Yaskawa INFORM job: OK_R2_O55B(90,0)KMOK.JBI

/JOB
//NAME OK_R2_O55B(90,0)KMOK
//POS
///NPOS 391,391,391,17,0,0
///TOOL 0
///POSTYPE PULSE
///PULSE
C00000=-9957,-80120,-66349,29251,62843,-41580
C00001=-130831,-56999,-52491,28072,65386,-40358
C00002=-127931,-24435,-32256,25248,67356,-37514
C00003=-126700,-19683,-26605,24973,66044,-37324
C00004=-125164,-19903,-26767,24398,65578,-36815
C00005=-126700,-19683,-26605,24973,66044,-37324
C00006=-126700,-19454,-24775,25160,65129,-37533
C00007=-126700,-19683,-26605,24973,66044,-37324
C00008=-126519,-14725,-22916,24857,66242,-37208
C00009=-126700,-19683,-26605,24973,66044,-37324
C00010=-127431,-22768,-30880,25062,67214,-37348
C00011=-129904,-26243,-35656,25771,69013,-37912
C00012=-103883,-33865,-42899,-26333,63628,-24210
C00013=-104076,-28068,-33208,-26929,60884,-23597
C00014=-104308,-24022,-28158,-27086,59888,-23435
C00015=-104293,-23807,-26929,-27261,59318,-23277
C00016=-104308,-24022,-28158,-27086,59888,-23435
C00017=-104568,-21372,-26276,-26919,59985,-23573
C00018=-104308,-24022,-28158,-27086,59888,-23435
C00019=-104359,-30091,-33838,-26967,60209,-23541
C00020=-104172,-35756,-40489,-26759,61329,-23752
C00021=-101371,-58624,-53351,-28997,58954,-21848
C00022=-130278,-21019,-10450,28766,57658,-40988
C00023=-127795,-16814,-4966,28257,55740,-40424
C00024=-124867,-3493,1682,21696,65206,-34879
C00025=-124867,-2956,3429,21830,64460,-35026
C00026=-124867,-3493,1682,21696,65206,-34879
C00027=-123403,-3637,1565,21295,64821,-34374
C00028=-124867,-3493,1682,21696,65206,-34879
C00029=-124781,112,4661,21670,65203,-34846
C00030=-126448,-16298,-3504,27965,54725,-40103
C00031=-127417,-18060,-5778,28164,55488,-40325
C00032=-129915,-24050,-16876,27962,59657,-40264
C00033=-103828,-30318,-23260,-29155,54504,-21694
C00034=-104023,-24208,-16094,-29514,53321,-21419
C00035=-104359,-18909,-9882,-29771,52240,-21236
C00036=-104359,-18502,-8615,-29989,51742,-21073
C00037=-104359,-18909,-9882,-29771,52240,-21236
C00038=-104548,-17165,-8596,-29647,52265,-21334
C00039=-104359,-18909,-9882,-29771,52240,-21236
C00040=-104284,-25793,-15917,-29738,52421,-21258
C00041=-104095,-31966,-23082,-29370,53571,-21532
C00042=-101389,-51580,-31391,-32519,50375,-19075
C00043=-130293,-20904,-10309,28779,57639,-41000
C00044=-127810,-16697,-4821,28272,55719,-40437
C00045=-124421,-5878,1074,22169,61673,-35261
C00046=-123293,-5978,993,21815,61369,-34862
C00047=-124421,-5878,1074,22169,61673,-35261
C00048=-124421,-5464,2370,22286,61130,-35375
C00049=-124421,-5878,1074,22169,61673,-35261
C00050=-124367,-3413,3070,22144,61694,-35234
C00051=-124421,-5878,1074,22169,61673,-35261
C00052=-127374,-17559,-5212,28177,55393,-40333
C00053=-129863,-23659,-16652,27928,59696,-40231
C00054=-104291,-30466,-23154,-28998,54219,-21823
C00055=-104471,-24344,-15984,-29365,53043,-21545
C00056=-104848,-18627,-9754,-29526,52126,-21437
C00057=-104848,-18034,-7918,-29844,51404,-21206
C00058=-104848,-18372,-8952,-29664,51809,-21336
C00059=-105025,-16673,-7696,-29545,51834,-21430
C00060=-104848,-18372,-8952,-29664,51809,-21336
C00061=-104541,-25679,-16044,-29572,52449,-21391
C00062=-104362,-31845,-23206,-29202,53599,-21667
C00063=-101422,-47913,-22789,-34118,47488,-17974
C00064=-130262,-20482,-9952,28769,57626,-40991
C00065=-127787,-16271,-4450,28267,55703,-40431
C00066=-125772,-1300,4566,24233,64800,-37238
C00067=-125099,-11874,382,27493,54175,-39643
C00068=-126165,-11734,491,27896,54532,-40029
C00069=-126165,-11290,1726,28071,54059,-40171
C00070=-126165,-11734,491,27896,54532,-40029
C00071=-126097,-9728,2048,27846,54574,-39985
C00072=-126165,-11734,491,27896,54532,-40029
C00073=-127493,-17714,-5356,28218,55441,-40373
C00074=-129987,-23980,-17397,27894,59998,-40203
C00075=-104210,-30109,-23029,-28998,54341,-21823
C00076=-104392,-23995,-15854,-29364,53158,-21544
C00077=-104664,-19137,-9875,-29681,52028,-21314
C00078=-104664,-18688,-8489,-29921,51485,-21138
C00079=-104664,-19137,-9875,-29681,52028,-21314
C00080=-104885,-17048,-8334,-29533,52061,-21432
C00081=-104664,-19137,-9875,-29681,52028,-21314
C00082=-104584,-25734,-15966,-29581,52368,-21386
C00083=-104406,-31905,-23130,-29210,53516,-21662
C00084=-101487,-56722,-46956,-29848,56320,-21116
C00085=-130260,-20245,-9571,28802,57525,-41018
C00086=-127787,-16027,-4057,28303,55600,-40460
C00087=-126397,-12024,-58,27921,54776,-40065
C00088=-126397,-11418,1630,28163,54132,-40255
C00089=-126397,-12024,-58,27921,54776,-40065
C00090=-125058,-12202,-195,27417,54327,-39580
C00091=-126397,-12024,-58,27921,54776,-40065
C00092=-126319,-9801,1666,27863,54821,-40014
C00093=-126397,-12024,-58,27921,54776,-40065
C00094=-127466,-17804,-5568,28181,55506,-40341
C00095=-129961,-24611,-19623,27616,60919,-39941
C00096=-104121,-29849,-22868,-29026,54402,-21800
C00097=-104306,-23738,-15686,-29392,53214,-21520
C00098=-104574,-18869,-9557,-29743,52009,-21266
C00099=-104574,-18451,-8267,-29970,51501,-21102
C00100=-104574,-18869,-9557,-29743,52009,-21266
C00101=-104772,-17011,-8185,-29613,52038,-21371
C00102=-104574,-18869,-9557,-29743,52009,-21266
C00103=-104605,-25690,-15920,-29574,52356,-21392
C00104=-101416,-53614,-36326,-31658,51963,-19708
C00105=-101416,-53614,-36326,-31658,51963,-19708
C00106=-113373,-19710,-23567,-5252,67661,-28636
C00107=-114752,-18608,-16975,3728,63450,-28918
C00108=-121641,-12158,-10795,16175,65821,-31343
C00109=-121641,-11553,-8404,16318,64706,-31501
C00110=-121642,-12221,-10110,16230,65385,-31404
C00111=-120492,-12233,-10119,15867,65157,-30993
C00112=-121644,-12965,-11195,16196,65660,-31365
C00113=-121703,-22742,-18426,16285,65120,-31465
C00114=-116423,-24349,-16589,8028,59581,-22849
C00115=-116462,-22943,-15594,8034,59695,-22855
C00116=-117089,-27968,-21523,8194,60813,-23017
C00117=-138257,-43921,-38980,29449,67834,19559
C00118=-154095,-44107,-36576,41026,64683,28586
C00119=-155372,-26710,-22710,49007,54658,45155
C00120=-156430,-13085,-10936,68207,72434,47480
C00121=-154097,-10834,-6257,68530,70189,47037
C00122=-153034,-8688,-2137,68930,68920,46537
C00123=-153034,-8230,-667,69164,68664,46234
C00124=-153034,-8688,-2137,68930,68920,46537
C00125=-152716,-7159,-923,68899,68723,46597
C00126=-153034,-8688,-2137,68930,68920,46537
C00127=-155527,-11962,-5672,68921,70786,46416
C00128=-157894,-14200,-10337,68577,73047,46860
C00129=-156589,-13315,-10824,68272,72466,47375
C00130=-154250,-11059,-6142,68601,70219,46932
C00131=-153110,-8549,-1740,68995,68901,46448
C00132=-153110,-8137,-433,69201,68672,46178
C00133=-153110,-8549,-1740,68995,68901,46448
C00134=-152772,-6933,-461,68963,68694,46512
C00135=-153110,-8549,-1740,68995,68901,46448
C00136=-155649,-11770,-5813,68871,70940,46483
C00137=-158013,-13984,-10461,68536,73200,46927
C00138=-156493,-13364,-11001,68241,72435,47426
C00139=-154155,-11109,-6321,68567,70188,46983
C00140=-153047,-8804,-2189,68941,68917,46522
C00141=-153047,-8341,-714,69171,68660,46216
C00142=-153047,-8804,-2189,68941,68917,46522
C00143=-152699,-7122,-856,68902,68699,46591
C00144=-153047,-8804,-2189,68941,68917,46522
C00145=-155528,-12235,-6032,68896,70818,46453
C00146=-157898,-14465,-10687,68556,73081,46895
C00147=-156404,-13719,-11255,68241,72365,47427
C00148=-154061,-11456,-6573,68567,70116,46985
C00149=-152978,-9293,-2613,68935,68873,46536
C00150=-152978,-8887,-1313,69141,68646,46265
C00151=-152978,-9293,-2613,68935,68873,46536
C00152=-152568,-7316,-1048,68891,68617,46616
C00153=-152978,-9293,-2613,68935,68873,46536
C00154=-155488,-12320,-6114,68891,70795,46461
C00155=-157860,-14552,-10769,68552,73058,46903
C00156=-156499,-13757,-11316,68244,72435,47421
C00157=-154155,-11502,-6641,68569,70186,46980
C00158=-152940,-8723,-2197,68919,68862,46557
C00159=-152940,-8321,-897,69127,68633,46287
C00160=-152940,-8723,-2197,68919,68862,46557
C00161=-152615,-7149,-950,68886,68660,46620
C00162=-152940,-8723,-2197,68919,68862,46557
C00163=-155527,-12441,-6175,68901,70811,46445
C00164=-157901,-14672,-10829,68562,73075,46886
C00165=-154973,1945,11064,69380,67800,43696
C00166=-153498,388,9750,69327,66810,43901
C00167=-151944,3598,13389,69509,65547,43839
C00168=-152901,-833,7436,68993,66712,44352
C00169=-153760,-1170,8451,69337,66987,43865
C00170=-150992,-308,10136,69473,64908,43968
C00171=-151435,4354,14125,69671,69854,43018
C00172=-151601,9028,18225,69679,74023,42144
C00173=-153599,495,9837,69084,71042,58093
C00174=-155601,2650,11659,69106,72383,57818
C00175=-155003,-799,3033,68136,69188,45300
C00176=-153529,-1129,5762,68693,67473,44668
C00177=-151691,2413,10794,69105,65750,44340
C00178=-152932,-1773,5149,68640,67090,44774
C00179=-153793,-2147,6130,68987,67361,44287
C00180=-151088,-288,8615,69107,65323,44406
C00181=-151404,3599,11904,69364,69896,43458
C00182=-151218,5876,13928,69450,72821,42839
C00183=-153630,-777,6611,68687,71576,58686
C00184=-155633,219,4703,68296,73580,59159
C00185=-154938,2214,11292,69379,67776,43700
C00186=-153465,658,9976,69326,66788,43906
C00187=-151970,3515,13352,69518,65553,43829
C00188=-152869,-564,7660,68991,66691,44357
C00189=-153727,-902,8674,69336,66964,43870
C00190=-151411,1015,11233,69490,65183,43915
C00191=-150298,-2919,8029,69467,64414,44045
C00192=-151641,9147,18309,69679,73942,42091
C00193=-153566,764,10064,69084,71020,58097
C00194=-155565,2919,11887,69107,72358,57821
C00195=-154990,1810,10950,69380,67812,43694
C00196=-153514,253,9637,69328,66822,43899
C00197=-151956,3103,12633,69423,65630,43940
C00198=-152917,-967,7324,68994,66723,44350
C00199=-153777,-1304,8340,69338,66998,43862
C00200=-151252,489,10575,69428,65130,44000
C00201=-151705,5965,15347,69658,70903,42778
C00202=-151762,10642,19506,69646,75062,41892
C00203=-153615,360,9724,69084,71054,58091
C00204=-155619,2515,11544,69106,72395,57816
C00205=-154955,2080,11178,69379,67788,43698
C00206=-153481,523,9864,69327,66799,43904
C00207=-152005,3278,13000,69479,65609,43868
C00208=-152885,-698,7548,68992,66701,44355
C00209=-153744,-1035,8563,69337,66975,43867
C00210=-151366,800,11018,69477,65161,43933
C00211=-151607,5013,14724,69679,69923,42916
C00212=-151807,11049,20057,69670,75075,41824
C00213=-153582,630,9951,69084,71031,58095
C00214=-155583,2785,11773,69106,72370,57820
C00215=-147758,2086,2374,31053,60988,58888
C00216=-133325,-38773,-33930,6315,58066,25890
C00217=-110400,-54315,-51528,-18458,56734,4707
C00218=-102274,-32558,-14872,-44027,37469,-32506
C00219=-105929,-26421,-10740,-41149,36164,-34321
C00220=-116067,-24319,-8645,-13286,26575,-50151
C00221=-116038,-24316,-8643,-13324,26580,-50130
C00222=-111352,-27223,-10659,-19551,27279,-46780
C00223=-103129,-25181,-9190,-38570,34106,-35952
C00224=-100769,-25035,-8960,-40367,35121,-34847
C00225=-99695,-24670,-8429,-41242,35512,-34306
C00226=-108656,-29084,-11659,-12032,25827,-50837
C00227=-110509,-34586,-17055,-9270,26069,-52303
C00228=-103616,-10758,2035,-15955,56275,-10509
C00229=-130330,-13924,-1675,30108,58090,-56546
C00230=-127978,-14439,-2068,29368,57239,-55742
C00231=-123256,-13385,-2249,22880,55912,-53736
C00232=-128068,-14313,-1975,29395,57277,-55771
C00233=-127033,-15220,-3955,28826,57580,-55217
C00234=-123207,-12197,-1342,22849,55945,-53708
C00235=-123090,-5999,3422,22738,56146,-53613
C00236=-123012,-3644,5328,22699,56159,-53576
C00237=-126427,-14696,-2262,28719,52056,-54431
C00238=-128721,-14290,-1952,29651,52868,-55271
C00239=-129847,-30322,-13664,30386,52393,-55913
C00240=-98615,-62310,-46614,-42670,42504,-33138
C00241=-102218,-38584,-32729,-38015,43544,-36056
C00242=-102480,-32544,-25881,-38582,42546,-35707
C00243=-103251,-25592,-19070,-38522,41713,-35751
C00244=-102756,-32211,-24481,-38883,41877,-35526
C00245=-102580,-30549,-24640,-38344,42709,-35853
C00246=-104239,-25243,-18850,-37852,41310,-36163
C00247=-105283,-24858,-18584,-37135,40880,-36603
C00248=-106143,-24446,-18295,-36529,40538,-36972
C00249=-106553,-24250,-18143,-36243,40369,-37147
C00250=-108719,-32876,-26099,-30904,38097,-40301
C00251=-108855,-38938,-32951,-30097,39002,-40766
C00252=-112694,-21246,-36478,-4917,71223,-21092
C00253=-111752,-21064,-33430,-5337,69507,-20687
C00254=-111684,-17344,-28816,-5396,68587,-20623
C00255=-111376,-20974,-33443,-5482,69586,-20557
C00256=-111534,-23106,-33731,-5452,68661,-20571
C00257=-110553,-17266,-28688,-5840,68626,-20217
C00258=-109244,-17338,-28705,-6354,68698,-19755
C00259=-108064,-17505,-28819,-6813,68777,-19334
C00260=-107309,-17780,-29023,-7104,68827,-19067
C00261=-104240,-18422,-31467,-13738,72317,-12857
C00262=-104358,-19286,-32232,-13695,72324,-12900
C00263=-130325,-20800,-32009,26820,71494,-52967
C00264=-127971,-21169,-29521,26293,69202,-52588
C00265=-125862,-20132,-27060,24855,67183,-52285
C00266=-128061,-20931,-28246,26431,68634,-52758
C00267=-127025,-21362,-29804,25958,68974,-52267
C00268=-125707,-18776,-26048,24786,67205,-52219
C00269=-125464,-12189,-21131,24639,67457,-52067
C00270=-125255,-10131,-19523,24550,67457,-51982
C00271=-126422,-21235,-27665,25246,63063,-51474
C00272=-128718,-21076,-30208,25849,65259,-51889
C00273=-129622,-34639,-39831,26336,64628,-52369
C00274=-100138,-47584,-24431,-46943,37343,-30712
C00275=-102344,-32235,-14659,-43953,37460,-32552
C00276=-102604,-27323,-11359,-43355,37695,-32905
C00277=-103274,-20911,-5782,-43063,37269,-33108
C00278=-102879,-27387,-11402,-43193,37556,-33012
C00279=-102702,-25990,-11742,-42495,38332,-33401
C00280=-104567,-20474,-5468,-42216,36668,-33654
C00281=-105669,-20033,-5149,-41463,36168,-34133
C00282=-106596,-19629,-4856,-40810,35756,-34545
C00283=-108815,-27628,-11564,-35628,32785,-37707
C00284=-108952,-32553,-14865,-35969,32319,-37533
C00285=-112746,-14120,-1833,-5728,53633,-20286
C00286=-111808,-13902,-1672,-6149,53715,-19902
C00287=-111460,-9500,2711,-6340,53311,-19729
C00288=-111434,-14423,-3365,-6257,54513,-19795
C00289=-111592,-15875,-3158,-6254,53633,-19807
C00290=-110314,-9638,2672,-6858,53358,-19256
C00291=-108552,-9905,2463,-7645,53507,-18533
C00292=-107785,-9902,2464,-7985,53582,-18217
C00293=-107177,-9829,2520,-8253,53644,-17968
C00294=-103878,-11141,478,-15725,56958,-10722
C00295=-105011,-11099,1638,-15418,56074,-11058
C00296=-130334,-13653,-1469,30106,58102,-56544
C00297=-127986,-14168,-1863,29367,57254,-55742
C00298=-121092,-13671,-3468,18618,55785,-52671
C00299=-128076,-14043,-1770,29394,57291,-55771
C00300=-127043,-14950,-3751,28825,57595,-55217
C00301=-124608,-11431,283,25762,55964,-54442
C00302=-124378,-5275,5018,25608,56118,-54300
C00303=-124320,-2361,7362,25553,56152,-54264
C00304=-126423,-14429,-2060,28712,52067,-54426
C00305=-128713,-14023,-1750,29643,52877,-55264
C00306=-131254,-24475,-9655,30465,57998,-56942
C00307=-100144,-47164,-24188,-46877,37386,-30750
C00308=-102238,-32719,-14978,-44064,37474,-32483
C00309=-102503,-27810,-11693,-43456,37711,-32843
C00310=-103289,-21357,-6334,-42954,37342,-33170
C00311=-102779,-27875,-11736,-43294,37571,-32950
C00312=-102603,-26479,-12082,-42592,38348,-33341
C00313=-104301,-20961,-6025,-42305,36863,-33590
C00314=-105481,-20525,-5713,-41507,36325,-34099
C00315=-106082,-20161,-5420,-41097,36048,-34359
C00316=-106580,-19948,-5267,-40743,35827,-34582
C00317=-108736,-28128,-11906,-35737,32779,-37645
C00318=-108871,-33052,-15192,-36089,32308,-37465
C00319=-112696,-16399,-7797,-5581,56123,-20400
C00320=-111755,-14868,-3629,-6120,54423,-19921
C00321=-111562,-9918,2203,-6286,53400,-19781
C00322=-111378,-14819,-3673,-6283,54504,-19771
C00323=-111536,-16269,-3462,-6281,53622,-19783
C00324=-110339,-10109,2128,-6839,53445,-19276
C00325=-109146,-10161,2155,-7376,53506,-18782
C00326=-108067,-10135,2207,-7857,53590,-18342
C00327=-107119,-10093,2237,-8275,53687,-17956
C00328=-105657,-13339,-2467,-12869,56371,-13559
C00329=-104122,-15984,-6399,-15346,58595,-11062
C00330=-130328,-14059,-1778,30110,58083,-56547
C00331=-127974,-14574,-2170,29369,57232,-55742
C00332=-126213,-11937,765,28926,56229,-55246
C00333=-128064,-14449,-2077,29396,57270,-55772
C00334=-127028,-15356,-4057,28827,57572,-55217
C00335=-126152,-10926,1517,28887,56258,-55209
C00336=-125945,-6265,5128,28761,56338,-55091
C00337=-125791,-2372,8223,28679,56370,-55012
C00338=-126392,-14836,-2368,28706,52039,-54420
C00339=-128688,-14432,-2060,29640,52851,-55260
C00340=-129555,-26680,-11188,30139,52591,-55707
C00341=-100121,-47554,-24413,-46948,37355,-30708
C00342=-102309,-32396,-14765,-43990,37465,-32529
C00343=-102570,-27485,-11470,-43388,37700,-32885
C00344=-103345,-21072,-5970,-42996,37257,-33150
C00345=-102846,-27550,-11513,-43226,37561,-32992
C00346=-102669,-26152,-11855,-42527,38337,-33381
C00347=-104275,-20857,-5845,-42378,36833,-33550
C00348=-105438,-20437,-5542,-41592,36301,-34053
C00349=-106155,-19944,-5110,-41121,35953,-34354
C00350=-106620,-19753,-4970,-40792,35747,-34561
C00351=-108789,-27794,-11678,-35664,32783,-37686
C00352=-108925,-32719,-14974,-36009,32315,-37511
C00353=-112729,-14250,-1932,-5737,53628,-20278
C00354=-111790,-14032,-1771,-6158,53710,-19894
C00355=-111584,-9413,2808,-6285,53286,-19783
C00356=-111416,-14553,-3463,-6266,54508,-19787
C00357=-111573,-16004,-3255,-6263,53627,-19799
C00358=-110680,-9603,2689,-6694,53333,-19410
C00359=-109622,-9847,2483,-7169,53423,-18977
C00360=-108783,-9926,2421,-7545,53497,-18631
C00361=-108041,-10006,2359,-7874,53566,-18327
C00362=-107142,-9915,2430,-8270,53659,-17959
C00363=-105001,-12679,-746,-13746,55987,-12713
C00364=-106768,-17459,-5146,-13005,55940,-13436
C00365=-130332,-13788,-1572,30107,58096,-56545
C00366=-127982,-14303,-1965,29368,57246,-55742
C00367=-126236,-11905,859,28945,56199,-55263
C00368=-128072,-14178,-1872,29395,57284,-55771
C00369=-127038,-15085,-3853,28826,57588,-55217
C00370=-126148,-10650,1810,28896,56222,-55217
C00371=-125895,-4713,6467,28751,56299,-55080
C00372=-125819,-1913,8722,28709,56319,-55040
C00373=-126436,-14560,-2159,28720,52065,-54433
C00374=-128728,-14154,-1848,29651,52876,-55272
C00375=-132513,-43218,-24407,28766,58278,-55899
C00376=-132513,-43218,-24407,28766,58278,-55899
C00377=-121666,-20715,-7127,19986,55197,-51612
C00378=-122063,-20657,-8381,19954,56049,-51613
C00379=-123700,-19829,-6494,20751,55763,-52369
C00380=-121964,-19403,-6177,20082,55352,-51709
C00381=-121700,-9961,769,19844,55835,-51502
C00382=-124810,-28520,-15259,20953,56913,-52609
C00383=-94216,-20206,-10160,-43887,70164,-41315
C00384=-105043,3978,10493,-37408,70381,-43017
C00385=-107559,8140,15454,-35830,70406,-43107
C00386=-111804,-1876,2679,-18365,65301,-43780
C00387=-109352,-1568,2008,-12034,65341,-42990
C00388=-109570,-19484,-5252,-8248,46858,-41038
C00389=-110437,-19763,-19574,-8377,68704,-43695
C00390=-141635,-113265,-78777,26632,71297,-57409
BC00000=15,674025,1075175
BC00001=16,674026,1075174
BC00002=15,674025,1075175
BC00003=15,674025,1075175
BC00004=16,674025,1075174
BC00005=15,674025,1075175
BC00006=15,674025,1075175
BC00007=15,674025,1075175
BC00008=15,674025,1075175
BC00009=15,674025,1075175
BC00010=15,674025,1075175
BC00011=15,674025,1075175
BC00012=15,675429,1075175
BC00013=15,675429,1075175
BC00014=15,675429,1075175
BC00015=15,675429,1075175
BC00016=15,675429,1075175
BC00017=15,675429,1075175
BC00018=15,675429,1075175
BC00019=15,675429,1075175
BC00020=15,675429,1075175
BC00021=15,675429,1075175
BC00022=15,675679,1044560
BC00023=15,675679,1044560
BC00024=15,675679,1044560
BC00025=15,675679,1044560
BC00026=15,675679,1044560
BC00027=15,675679,1044560
BC00028=15,675679,1044560
BC00029=15,675679,1044560
BC00030=15,675679,1044560
BC00031=15,675679,1044560
BC00032=15,675679,1044560
BC00033=15,675432,1006215
BC00034=15,675432,1006215
BC00035=15,675432,1006215
BC00036=15,675432,1006215
BC00037=15,675432,1006215
BC00038=15,675432,1006215
BC00039=15,675432,1006215
BC00040=15,675432,1006215
BC00041=15,675432,1006215
BC00042=15,675429,1028113
BC00043=15,675400,880877
BC00044=15,675400,880877
BC00045=15,675400,880877
BC00046=15,675400,880877
BC00047=15,675400,880877
BC00048=15,675400,880877
BC00049=15,675400,880877
BC00050=15,675400,880877
BC00051=15,675400,880877
BC00052=15,675400,880877
BC00053=15,675400,880877
BC00054=15,675485,845406
BC00055=15,675485,845406
BC00056=15,675485,845406
BC00057=15,675485,845406
BC00058=15,675485,845406
BC00059=15,675485,845406
BC00060=15,675485,845406
BC00061=15,675485,845406
BC00062=15,675485,845406
BC00063=15,675429,906681
BC00064=15,675816,718619
BC00065=15,675816,718619
BC00066=15,675816,718619
BC00067=15,675816,718619
BC00068=15,675816,718619
BC00069=15,675816,718619
BC00070=15,675816,718619
BC00071=15,675816,718619
BC00072=15,675816,718619
BC00073=15,675816,718619
BC00074=15,675816,718619
BC00075=15,675806,682567
BC00076=15,675806,682567
BC00077=15,675806,682567
BC00078=15,675806,682567
BC00079=15,675806,682567
BC00080=15,675806,682567
BC00081=15,675806,682567
BC00082=15,675806,682567
BC00083=15,675806,682567
BC00084=15,675429,625602
BC00085=15,676009,556911
BC00086=15,676009,556911
BC00087=15,676009,556911
BC00088=15,676009,556911
BC00089=15,676009,556911
BC00090=15,676009,556911
BC00091=15,676009,556911
BC00092=15,676009,556911
BC00093=15,676009,556911
BC00094=15,676009,556911
BC00095=15,676009,556911
BC00096=15,675951,521174
BC00097=15,675951,521174
BC00098=15,675951,521174
BC00099=15,675951,521174
BC00100=15,675951,521174
BC00101=15,675951,521174
BC00102=15,675951,521174
BC00103=15,675951,521174
BC00104=15,675951,521174
BC00105=15,675951,304544
BC00106=15,675951,304544
BC00107=15,675951,304544
BC00108=15,675951,304544
BC00109=15,675951,304544
BC00110=15,675951,304544
BC00111=15,675951,304544
BC00112=15,675951,304544
BC00113=15,675951,304544
BC00114=15,675951,304544
BC00115=15,675951,304544
BC00116=15,675951,304544
BC00117=15,683095,452911
BC00118=15,684575,438764
BC00119=15,686333,421965
BC00120=15,687857,407402
BC00121=15,687857,407402
BC00122=15,687857,407402
BC00123=15,687857,407402
BC00124=15,687857,407402
BC00125=15,687857,407402
BC00126=15,687857,407402
BC00127=15,687857,407402
BC00128=15,687857,407402
BC00129=15,687790,570534
BC00130=15,687790,570534
BC00131=15,687790,570534
BC00132=15,687790,570534
BC00133=15,687790,570534
BC00134=15,687790,570534
BC00135=15,687790,570534
BC00136=15,687790,570534
BC00137=15,687790,570534
BC00138=15,687643,731759
BC00139=15,687643,731759
BC00140=15,687643,731759
BC00141=15,687643,731759
BC00142=15,687643,731759
BC00143=15,687643,731759
BC00144=15,687643,731759
BC00145=15,687643,731759
BC00146=15,687643,731759
BC00147=15,687421,893970
BC00148=15,687421,893970
BC00149=15,687421,893970
BC00150=15,687421,893970
BC00151=15,687421,893970
BC00152=15,687421,893970
BC00153=15,687421,893970
BC00154=15,687421,893970
BC00155=15,687421,893970
BC00156=15,687425,1055071
BC00157=15,687425,1055071
BC00158=15,687425,1055071
BC00159=15,687425,1055071
BC00160=15,687425,1055071
BC00161=15,687425,1055071
BC00162=15,687425,1055071
BC00163=15,687425,1055071
BC00164=15,687425,1055071
BC00165=15,675237,787703
BC00166=15,679011,768774
BC00167=15,680512,761248
BC00168=15,680521,761203
BC00169=15,680521,761203
BC00170=15,680521,761203
BC00171=15,680521,761203
BC00172=15,680521,761203
BC00173=15,682227,765270
BC00174=15,679811,782503
BC00175=15,675146,1075175
BC00176=15,678921,1075175
BC00177=15,680430,1075172
BC00178=15,680430,1075175
BC00179=15,680430,1075175
BC00180=16,680430,1075169
BC00181=16,680430,1075169
BC00182=16,680430,1075169
BC00183=15,682137,1075175
BC00184=15,679720,1075175
BC00185=15,675327,464292
BC00186=15,679101,445363
BC00187=15,680611,437792
BC00188=15,680611,437792
BC00189=15,680611,437792
BC00190=15,680611,437792
BC00191=15,680611,437792
BC00192=15,680611,437792
BC00193=15,682318,441859
BC00194=15,679901,459092
BC00195=15,675192,949812
BC00196=15,678966,930883
BC00197=15,680476,923311
BC00198=15,680476,923311
BC00199=15,680476,923311
BC00200=15,680476,923311
BC00201=15,680476,923311
BC00202=15,680476,923311
BC00203=15,682182,927378
BC00204=15,679765,944612
BC00205=15,675282,625594
BC00206=15,679056,606665
BC00207=15,680566,599094
BC00208=15,680566,599094
BC00209=15,680566,599094
BC00210=15,680566,599094
BC00211=15,680566,599094
BC00212=15,680566,599094
BC00213=15,682273,603161
BC00214=15,679856,620394
BC00215=15,677299,661477
BC00216=15,673454,723260
BC00217=15,670450,771529
BC00218=15,666220,839502
BC00219=15,666220,820793
BC00220=15,666220,813310
BC00221=15,666220,813310
BC00222=15,666220,813310
BC00223=15,666220,813310
BC00224=15,666220,813310
BC00225=15,666220,813310
BC00226=15,666220,813310
BC00227=15,666220,813310
BC00228=15,667710,939573
BC00229=15,670096,912804
BC00230=15,672475,894941
BC00231=15,673427,887796
BC00232=15,673427,887796
BC00233=15,673427,887796
BC00234=15,673427,887796
BC00235=15,673427,887796
BC00236=15,673427,887796
BC00237=15,670651,882623
BC00238=15,667644,899848
BC00239=15,667644,899848
BC00240=15,666220,1075175
BC00241=15,666220,1075175
BC00242=15,666220,1075175
BC00243=15,666220,1075175
BC00244=15,666220,1075175
BC00245=15,666220,1075175
BC00246=15,666220,1075175
BC00247=15,666220,1075175
BC00248=15,666220,1075175
BC00249=15,666220,1075175
BC00250=15,666220,1075175
BC00251=15,666220,1075175
BC00252=15,669501,1075175
BC00253=15,674544,1075175
BC00254=15,676561,1075175
BC00255=15,676561,1075175
BC00256=15,676561,1075175
BC00257=15,676561,1075175
BC00258=15,676561,1075175
BC00259=15,676561,1075175
BC00260=15,676561,1075175
BC00261=15,672972,1075175
BC00262=15,667619,1075175
BC00263=15,670005,1075175
BC00264=15,672385,1075175
BC00265=15,673337,1075175
BC00266=15,673337,1075175
BC00267=15,673337,1075175
BC00268=15,673337,1075175
BC00269=15,673337,1075175
BC00270=15,673337,1075175
BC00271=15,670408,1075175
BC00272=15,667401,1075175
BC00273=15,667401,1075175
BC00274=15,666220,516091
BC00275=15,666220,516091
BC00276=15,666220,497382
BC00277=15,666220,489899
BC00278=15,666220,489899
BC00279=15,666220,489899
BC00280=15,666220,489899
BC00281=15,666220,489899
BC00282=15,666220,489899
BC00283=15,666220,497395
BC00284=15,666220,516103
BC00285=15,669682,616208
BC00286=15,674724,597282
BC00287=15,676741,589712
BC00288=15,676741,589712
BC00289=15,676741,589712
BC00290=15,676741,589712
BC00291=15,676741,589712
BC00292=15,676741,589712
BC00293=15,676741,589712
BC00294=15,673153,597239
BC00295=15,667800,616162
BC00296=15,670186,589392
BC00297=15,672565,571530
BC00298=15,673517,564385
BC00299=15,673517,564385
BC00300=15,673517,564385
BC00301=15,673517,564385
BC00302=15,673517,564385
BC00303=16,673517,564382
BC00304=15,671355,559209
BC00305=15,668348,576434
BC00306=15,670186,589392
BC00307=15,666220,1001611
BC00308=15,666220,1001611
BC00309=15,666220,982902
BC00310=15,666220,975418
BC00311=15,666220,975418
BC00312=15,666220,975418
BC00313=15,666220,975418
BC00314=15,666220,975418
BC00315=15,666220,975418
BC00316=15,666220,975418
BC00317=15,666220,982914
BC00318=15,666220,1001623
BC00319=15,669546,1075175
BC00320=15,674589,1075175
BC00321=15,676606,1075175
BC00322=15,676606,1075175
BC00323=15,676606,1075175
BC00324=15,676606,1075175
BC00325=15,676606,1075175
BC00326=15,676606,1075175
BC00327=15,676606,1075175
BC00328=15,673017,1075175
BC00329=15,667665,1075175
BC00330=15,670050,1074912
BC00331=15,672430,1057050
BC00332=15,673382,1049905
BC00333=15,673382,1049905
BC00334=15,673382,1049905
BC00335=15,673382,1049905
BC00336=15,673382,1049905
BC00337=15,673382,1049905
BC00338=15,671837,1044726
BC00339=15,668831,1061952
BC00340=15,668831,1061952
BC00341=15,666220,677393
BC00342=15,666220,677393
BC00343=15,666220,658684
BC00344=15,666220,651201
BC00345=15,666220,651201
BC00346=15,666220,651201
BC00347=15,666220,651201
BC00348=15,666220,651201
BC00349=15,666220,651201
BC00350=15,666220,651201
BC00351=15,666220,658697
BC00352=15,666220,677405
BC00353=15,669637,777510
BC00354=15,674679,758584
BC00355=15,676696,751014
BC00356=15,676696,751014
BC00357=15,676696,751014
BC00358=15,676696,751014
BC00359=15,676696,751014
BC00360=15,676696,751014
BC00361=15,676696,751014
BC00362=15,676696,751014
BC00363=15,673108,758541
BC00364=15,673108,758541
BC00365=15,670141,750695
BC00366=15,672520,732832
BC00367=15,673472,725687
BC00368=15,673472,725687
BC00369=15,673472,725687
BC00370=15,673472,725687
BC00371=15,673472,725687
BC00372=15,673472,725687
BC00373=15,670543,720515
BC00374=15,667536,737740
BC00375=15,668300,741539
BC00376=15,681177,346578
BC00377=15,681177,346578
BC00378=15,681177,346578
BC00379=15,681177,346578
BC00380=15,681177,346578
BC00381=15,681177,346578
BC00382=15,681177,346578
BC00383=15,681177,346578
BC00384=15,681177,346578
BC00385=15,681177,346578
BC00386=15,681177,346578
BC00387=15,681177,346578
BC00388=15,681177,346578
BC00389=15,681177,346578
BC00390=15,670141,750695
EC00000=798156,0
EC00001=798153,2
EC00002=798156,0
EC00003=798156,0
EC00004=798155,0
EC00005=798156,0
EC00006=798156,0
EC00007=798156,0
EC00008=798156,0
EC00009=798156,0
EC00010=798156,0
EC00011=798156,0
EC00012=798156,0
EC00013=798156,0
EC00014=798156,0
EC00015=798156,0
EC00016=798156,0
EC00017=798156,0
EC00018=798156,0
EC00019=798156,0
EC00020=798156,0
EC00021=798156,0
EC00022=798156,0
EC00023=798156,0
EC00024=798156,0
EC00025=798156,0
EC00026=798156,0
EC00027=798156,0
EC00028=798156,0
EC00029=798156,0
EC00030=798156,0
EC00031=798156,0
EC00032=798156,0
EC00033=798156,0
EC00034=798156,0
EC00035=798156,0
EC00036=798156,0
EC00037=798156,0
EC00038=798156,0
EC00039=798156,0
EC00040=798156,0
EC00041=798156,0
EC00042=798156,0
EC00043=798156,0
EC00044=798156,0
EC00045=798156,0
EC00046=798156,0
EC00047=798156,0
EC00048=798156,0
EC00049=798156,0
EC00050=798156,0
EC00051=798156,0
EC00052=798156,0
EC00053=798156,0
EC00054=798156,0
EC00055=798156,0
EC00056=798156,0
EC00057=798156,0
EC00058=798156,0
EC00059=798156,0
EC00060=798156,0
EC00061=798156,0
EC00062=798156,0
EC00063=798156,0
EC00064=798156,0
EC00065=798156,0
EC00066=798156,0
EC00067=798156,0
EC00068=798156,0
EC00069=798156,0
EC00070=798156,0
EC00071=798156,0
EC00072=798156,0
EC00073=798156,0
EC00074=798156,0
EC00075=798156,0
EC00076=798156,0
EC00077=798156,0
EC00078=798156,0
EC00079=798156,0
EC00080=798156,0
EC00081=798156,0
EC00082=798156,0
EC00083=798156,0
EC00084=798156,0
EC00085=798156,0
EC00086=798156,0
EC00087=798156,0
EC00088=798156,0
EC00089=798156,0
EC00090=798156,0
EC00091=798156,0
EC00092=798156,0
EC00093=798156,0
EC00094=798156,0
EC00095=798156,0
EC00096=798156,0
EC00097=798156,0
EC00098=798156,0
EC00099=798156,0
EC00100=798156,0
EC00101=798156,0
EC00102=798156,0
EC00103=798156,0
EC00104=798156,0
EC00105=798156,0
EC00106=798156,0
EC00107=798156,0
EC00108=798156,0
EC00109=798156,0
EC00110=798156,0
EC00111=798156,0
EC00112=798156,0
EC00113=798156,0
EC00114=798156,0
EC00115=798156,0
EC00116=798156,0
EC00117=798156,0
EC00118=798156,0
EC00119=798156,0
EC00120=798156,0
EC00121=798156,0
EC00122=798156,0
EC00123=798156,0
EC00124=798156,0
EC00125=798156,0
EC00126=798156,0
EC00127=798156,0
EC00128=798156,0
EC00129=798156,0
EC00130=798156,0
EC00131=798156,0
EC00132=798156,0
EC00133=798156,0
EC00134=798156,0
EC00135=798156,0
EC00136=798156,0
EC00137=798156,0
EC00138=798156,0
EC00139=798156,0
EC00140=798156,0
EC00141=798156,0
EC00142=798156,0
EC00143=798156,0
EC00144=798156,0
EC00145=798156,0
EC00146=798156,0
EC00147=798156,0
EC00148=798156,0
EC00149=798156,0
EC00150=798156,0
EC00151=798156,0
EC00152=798156,0
EC00153=798156,0
EC00154=798156,0
EC00155=798156,0
EC00156=798156,0
EC00157=798156,0
EC00158=798156,0
EC00159=798156,0
EC00160=798156,0
EC00161=798156,0
EC00162=798156,0
EC00163=798156,0
EC00164=798156,0
EC00165=798156,0
EC00166=798156,0
EC00167=798156,0
EC00168=798156,0
EC00169=798156,0
EC00170=798156,0
EC00171=798156,0
EC00172=798156,0
EC00173=798156,0
EC00174=798156,0
EC00175=798156,0
EC00176=798156,0
EC00177=798155,0
EC00178=798156,0
EC00179=798156,0
EC00180=798154,1
EC00181=798154,1
EC00182=798154,1
EC00183=798156,0
EC00184=798156,0
EC00185=798156,0
EC00186=798156,0
EC00187=798156,0
EC00188=798156,0
EC00189=798156,0
EC00190=798156,0
EC00191=798156,0
EC00192=798156,0
EC00193=798156,0
EC00194=798156,0
EC00195=798156,0
EC00196=798156,0
EC00197=798156,0
EC00198=798156,0
EC00199=798156,0
EC00200=798156,0
EC00201=798156,0
EC00202=798156,0
EC00203=798156,0
EC00204=798156,0
EC00205=798156,0
EC00206=798156,0
EC00207=798156,0
EC00208=798156,0
EC00209=798156,0
EC00210=798156,0
EC00211=798156,0
EC00212=798156,0
EC00213=798156,0
EC00214=798156,0
EC00215=798156,0
EC00216=798156,0
EC00217=798156,0
EC00218=798156,0
EC00219=798156,0
EC00220=798156,0
EC00221=798156,0
EC00222=798156,0
EC00223=798156,0
EC00224=798156,0
EC00225=798156,0
EC00226=798156,0
EC00227=798156,0
EC00228=798156,0
EC00229=798156,0
EC00230=798156,0
EC00231=798156,0
EC00232=798156,0
EC00233=798156,0
EC00234=798156,0
EC00235=798156,0
EC00236=798156,0
EC00237=798156,0
EC00238=798156,0
EC00239=798156,0
EC00240=798156,0
EC00241=798156,0
EC00242=798156,0
EC00243=798156,0
EC00244=798156,0
EC00245=798156,0
EC00246=798156,0
EC00247=798156,0
EC00248=798156,0
EC00249=798156,0
EC00250=798156,0
EC00251=798156,0
EC00252=798156,0
EC00253=798156,0
EC00254=798156,0
EC00255=798156,0
EC00256=798156,0
EC00257=798156,0
EC00258=798156,0
EC00259=798156,0
EC00260=798156,0
EC00261=798156,0
EC00262=798156,0
EC00263=798156,0
EC00264=798156,0
EC00265=798156,0
EC00266=798156,0
EC00267=798156,0
EC00268=798156,0
EC00269=798156,0
EC00270=798156,0
EC00271=798156,0
EC00272=798156,0
EC00273=798156,0
EC00274=798156,0
EC00275=798156,0
EC00276=798156,0
EC00277=798156,0
EC00278=798156,0
EC00279=798156,0
EC00280=798156,0
EC00281=798156,0
EC00282=798156,0
EC00283=798156,0
EC00284=798156,0
EC00285=798156,0
EC00286=798156,0
EC00287=798156,0
EC00288=798156,0
EC00289=798156,0
EC00290=798156,0
EC00291=798156,0
EC00292=798156,0
EC00293=798156,0
EC00294=798156,0
EC00295=798156,0
EC00296=798156,0
EC00297=798156,0
EC00298=798156,0
EC00299=798156,0
EC00300=798156,0
EC00301=798156,0
EC00302=798156,0
EC00303=798155,0
EC00304=798156,0
EC00305=798156,0
EC00306=798156,0
EC00307=798156,0
EC00308=798156,0
EC00309=798156,0
EC00310=798156,0
EC00311=798156,0
EC00312=798156,0
EC00313=798156,0
EC00314=798156,0
EC00315=798156,0
EC00316=798156,0
EC00317=798156,0
EC00318=798156,0
EC00319=798156,0
EC00320=798156,0
EC00321=798156,0
EC00322=798156,0
EC00323=798156,0
EC00324=798156,0
EC00325=798156,0
EC00326=798156,0
EC00327=798156,0
EC00328=798156,0
EC00329=798156,0
EC00330=798156,0
EC00331=798156,0
EC00332=798156,0
EC00333=798156,0
EC00334=798156,0
EC00335=798156,0
EC00336=798156,0
EC00337=798156,0
EC00338=798156,0
EC00339=798156,0
EC00340=798156,0
EC00341=798156,0
EC00342=798156,0
EC00343=798156,0
EC00344=798156,0
EC00345=798156,0
EC00346=798156,0
EC00347=798156,0
EC00348=798156,0
EC00349=798156,0
EC00350=798156,0
EC00351=798156,0
EC00352=798156,0
EC00353=798156,0
EC00354=798156,0
EC00355=798156,0
EC00356=798156,0
EC00357=798156,0
EC00358=798156,0
EC00359=798156,0
EC00360=798156,0
EC00361=798156,0
EC00362=798156,0
EC00363=798156,0
EC00364=798156,0
EC00365=798156,0
EC00366=798156,0
EC00367=798156,0
EC00368=798156,0
EC00369=798156,0
EC00370=798156,0
EC00371=798156,0
EC00372=798156,0
EC00373=798156,0
EC00374=798156,0
EC00375=798156,0
EC00376=798156,0
EC00377=798156,0
EC00378=798156,0
EC00379=798156,0
EC00380=798156,0
EC00381=798156,0
EC00382=798156,0
EC00383=798156,0
EC00384=798156,0
EC00385=798156,0
EC00386=798156,0
EC00387=798156,0
EC00388=798156,0
EC00389=798156,0
EC00390=798156,0
///POSTYPE BASE
///RECTAN
///RCONF 0,0,0,0,0,0,0,0,0,0,0,0,0,0,0,0,0,0,0,0,0,0,0,0
P00006=0.222,-3.123,-1.508,0.0000,0.0000,0.0000
P00021=-0.225,-6.128,-0.405,0.0000,0.0000,0.0000
P00022=0.222,-3.123,-1.508,0.0000,0.0000,0.0000
P00023=0.143,-0.036,0.682,0.0000,0.0000,0.0000
P00031=1.853,-0.001,-1.549,0.0000,0.0000,0.0000
P00032=1.957,0.503,-7.217,0.0000,0.0000,0.0000
///RCONF 0,0,0,0,1,0,0,0,0,0,0,0,0,0,0,0,0,0,0,0,0,0,0,0
P00033=-0.123,0.612,-5.012,0.0000,0.0000,0.0000
///RCONF 0,0,0,0,0,0,0,0,0,0,0,0,0,0,0,0,0,0,0,0,0,0,0,0
P00041=0.192,3.924,0.305,0.0000,0.0000,0.0000
P00042=-0.217,1.941,0.413,0.0000,0.0000,0.0000
P00043=-0.044,-1.937,1.197,0.0000,0.0000,0.0000
P00051=0.367,3.892,0.009,0.0000,0.0000,0.0000
P00052=0.088,2.832,-0.342,0.0000,0.0000,0.0000
P00053=0.134,6.594,0.107,0.0000,0.0000,0.0000
P00061=1.575,-3.405,-0.752,0.0000,0.0000,0.0000
P00062=-0.135,-0.848,-1.706,0.0000,0.0000,0.0000
P00063=0.036,-0.654,-3.005,0.0000,0.0000,0.0000
P00100=1.890,0.539,-2.641,0.0000,0.0000,0.0000
//INST
///DATE 2025/01/24 12:06
///ATTR SC,RW
///GROUP1 RB1,BS1
///GROUP2 ST1
NOP
'MUZYLO 310124
'POPRAWA I SPAWANIE
'OK_R2_o55b(90,0)
'
'Path S3809
SFTOF3D
MOVJ C00000 BC00000 VJ=100.00  +MOVJ EC00000 VJ=100.00
CALL JOB:CLEAN-R1_KM_NEW
MOVJ C00001 BC00001 VJ=100.00  +MOVJ EC00001 VJ=100.00
MOVL C00002 BC00002 V=666.7  +MOVJ EC00002 VJ=100.00
SMOVL C00003 BC00003 V=133.3  +MOVJ EC00003
SREFP 3 C00004 BC00004  +REFP EC00004
CALL JOB:SEARCH-R1-S13D
SET P021 P006
SFTON3D P021
SMOVL C00005 BC00005 V=166.7  +MOVJ EC00005
SREFP 3 C00006 BC00006  +REFP EC00006
CALL JOB:SEARCH-R1-S13D
SET P021 P006
SFTON3D P021
SMOVL C00007 BC00007 V=166.7  +MOVJ EC00007
SREFP 3 C00008 BC00008  +REFP EC00008
CALL JOB:SEARCH-R1-S13D
SET P021 P006
SFTON3D P021
SMOVL C00009 BC00009 V=166.7  +MOVJ EC00009
MOVL C00010 BC00010 V=666.7  +MOVJ EC00010 VJ=100.00
MOVL C00011 BC00011 V=1000.0  +MOVJ EC00011 VJ=100.00
'Path S3810
SFTOF3D
MOVJ C00012 BC00012 VJ=100.00  +MOVJ EC00012 VJ=100.00
MOVL C00013 BC00013 V=666.7  +MOVJ EC00013 VJ=100.00
SMOVL C00014 BC00014 V=133.3  +MOVJ EC00014
SREFP 3 C00015 BC00015  +REFP EC00015
CALL JOB:SEARCH-R1-S13D
SET P022 P006
SFTON3D P022
SMOVL C00016 BC00016 V=166.7  +MOVJ EC00016
SREFP 3 C00017 BC00017  +REFP EC00017
CALL JOB:SEARCH-R1-S13D
SET P022 P006
SFTON3D P022
SMOVL C00018 BC00018 V=166.7  +MOVJ EC00018
MOVL C00019 BC00019 V=666.7  +MOVJ EC00019 VJ=100.00
MOVL C00020 BC00020 V=1000.0  +MOVJ EC00020 VJ=100.00
MOVJ C00021 BC00021 VJ=100.00  +MOVJ EC00021 VJ=100.00
'
'Path S3811
SFTOF3D
MOVJ C00022 BC00022 VJ=100.00  +MOVJ EC00022 VJ=100.00
MOVL C00023 BC00023 V=666.7  +MOVJ EC00023 VJ=100.00
SMOVL C00024 BC00024 V=133.3  +MOVJ EC00024
SREFP 3 C00025 BC00025  +REFP EC00025
CALL JOB:SEARCH-R1-S13D
SET P031 P006
SFTON3D P031
SMOVL C00026 BC00026 V=166.7  +MOVJ EC00026
SREFP 3 C00027 BC00027  +REFP EC00027
CALL JOB:SEARCH-R1-S13D
SET P031 P006
SFTON3D P031
SMOVL C00028 BC00028 V=166.7  +MOVJ EC00028
SREFP 3 C00029 BC00029  +REFP EC00029
CALL JOB:SEARCH-R1-S13D
SET P031 P006
SFTON3D P031
SMOVL C00030 BC00030 V=166.7  +MOVJ EC00030
MOVL C00031 BC00031 V=666.7  +MOVJ EC00031 VJ=100.00
MOVL C00032 BC00032 V=1000.0  +MOVJ EC00032 VJ=100.00
'Path S3812
SFTOF3D
MOVJ C00033 BC00033 VJ=100.00  +MOVJ EC00033 VJ=100.00
MOVL C00034 BC00034 V=666.7  +MOVJ EC00034 VJ=100.00
SMOVL C00035 BC00035 V=166.7  +MOVJ EC00035
SREFP 3 C00036 BC00036  +REFP EC00036
CALL JOB:SEARCH-R1-S13D
SET P032 P006
SFTON3D P032
SMOVL C00037 BC00037 V=166.7  +MOVJ EC00037
SREFP 3 C00038 BC00038  +REFP EC00038
CALL JOB:SEARCH-R1-S13D
SET P032 P006
SFTON3D P032
SMOVL C00039 BC00039 V=166.7  +MOVJ EC00039
MOVL C00040 BC00040 V=666.7  +MOVJ EC00040 VJ=100.00
MOVL C00041 BC00041 V=1000.0  +MOVJ EC00041 VJ=100.00
MOVJ C00042 BC00042 VJ=100.00  +MOVJ EC00042 VJ=100.00
'
'Path S3813
SFTOF3D
MOVJ C00043 BC00043 VJ=100.00  +MOVJ EC00043 VJ=100.00
MOVL C00044 BC00044 V=666.7  +MOVJ EC00044 VJ=100.00
SMOVL C00045 BC00045 V=133.3  +MOVJ EC00045
SREFP 3 C00046 BC00046  +REFP EC00046
CALL JOB:SEARCH-R1-S13D
SET P041 P006
SFTON3D P041
SMOVL C00047 BC00047 V=133.3  +MOVJ EC00047
SREFP 3 C00048 BC00048  +REFP EC00048
CALL JOB:SEARCH-R1-S13D
SET P041 P006
SFTON3D P041
SMOVL C00049 BC00049 V=133.3  +MOVJ EC00049
SREFP 3 C00050 BC00050  +REFP EC00050
CALL JOB:SEARCH-R1-S13D
SET P041 P006
SFTON3D P041
SMOVL C00051 BC00051 V=166.7  +MOVJ EC00051
MOVL C00052 BC00052 V=666.7  +MOVJ EC00052 VJ=100.00
MOVL C00053 BC00053 V=1000.0  +MOVJ EC00053 VJ=100.00
'Path S3814
SFTOF3D
MOVJ C00054 BC00054 VJ=100.00  +MOVJ EC00054 VJ=100.00
MOVL C00055 BC00055 V=666.7  +MOVJ EC00055 VJ=100.00
SMOVL C00056 BC00056 V=133.3  +MOVJ EC00056
SREFP 3 C00057 BC00057  +REFP EC00057
CALL JOB:SEARCH-R1-S13D
SET P042 P006
SFTON3D P042
SMOVL C00058 BC00058 V=166.7  +MOVJ EC00058
SREFP 3 C00059 BC00059  +REFP EC00059
CALL JOB:SEARCH-R1-S13D
SET P042 P006
SFTON3D P042
SMOVL C00060 BC00060 V=166.7  +MOVJ EC00060
MOVL C00061 BC00061 V=666.7  +MOVJ EC00061 VJ=100.00
MOVL C00062 BC00062 V=1000.0  +MOVJ EC00062 VJ=100.00
MOVJ C00063 BC00063 VJ=100.00  +MOVJ EC00063 VJ=100.00
'
'Path S3815
SFTOF3D
MOVJ C00064 BC00064 VJ=100.00  +MOVJ EC00064 VJ=100.00
MOVL C00065 BC00065 V=666.7  +MOVJ EC00065 VJ=100.00
SMOVL C00066 BC00066 V=133.3  +MOVJ EC00066
SREFP 3 C00067 BC00067  +REFP EC00067
CALL JOB:SEARCH-R1-S13D
SET P051 P006
SFTON3D P051
SMOVL C00068 BC00068 V=166.7  +MOVJ EC00068
SREFP 3 C00069 BC00069  +REFP EC00069
CALL JOB:SEARCH-R1-S13D
SET P051 P006
SFTON3D P051
SMOVL C00070 BC00070 V=166.7  +MOVJ EC00070
SREFP 3 C00071 BC00071  +REFP EC00071
CALL JOB:SEARCH-R1-S13D
SET P051 P006
SFTON3D P051
SMOVL C00072 BC00072 V=166.7  +MOVJ EC00072
MOVL C00073 BC00073 V=666.7  +MOVJ EC00073 VJ=100.00
MOVL C00074 BC00074 V=1000.0  +MOVJ EC00074 VJ=100.00
'Path S3816
SFTOF3D
MOVJ C00075 BC00075 VJ=100.00  +MOVJ EC00075 VJ=100.00
MOVL C00076 BC00076 V=666.7  +MOVJ EC00076 VJ=100.00
SMOVL C00077 BC00077 V=133.3  +MOVJ EC00077
SREFP 3 C00078 BC00078  +REFP EC00078
CALL JOB:SEARCH-R1-S13D
SET P052 P006
SFTON3D P052
SMOVL C00079 BC00079 V=166.7  +MOVJ EC00079
SREFP 3 C00080 BC00080  +REFP EC00080
CALL JOB:SEARCH-R1-S13D
SET P052 P006
SFTON3D P052
SMOVL C00081 BC00081 V=166.7  +MOVJ EC00081
MOVL C00082 BC00082 V=666.7  +MOVJ EC00082 VJ=100.00
MOVL C00083 BC00083 V=1000.0  +MOVJ EC00083 VJ=100.00
MOVJ C00084 BC00084 VJ=100.00  +MOVJ EC00084 VJ=100.00
'
'Path S3817
SFTOF3D
MOVJ C00085 BC00085 VJ=100.00  +MOVJ EC00085 VJ=100.00
MOVL C00086 BC00086 V=666.7  +MOVJ EC00086 VJ=100.00
SMOVL C00087 BC00087 V=166.7  +MOVJ EC00087
SREFP 3 C00088 BC00088  +REFP EC00088
CALL JOB:SEARCH-R1-S13D
SET P061 P006
SFTON3D P061
SMOVL C00089 BC00089 V=166.7  +MOVJ EC00089
SREFP 3 C00090 BC00090  +REFP EC00090
CALL JOB:SEARCH-R1-S13D
SET P061 P006
SFTON3D P061
SMOVL C00091 BC00091 V=166.7  +MOVJ EC00091
SREFP 3 C00092 BC00092  +REFP EC00092
CALL JOB:SEARCH-R1-S13D
SET P061 P006
SFTON3D P061
SMOVL C00093 BC00093 V=166.7  +MOVJ EC00093
MOVL C00094 BC00094 V=666.7  +MOVJ EC00094 VJ=100.00
MOVL C00095 BC00095 V=1000.0  +MOVJ EC00095 VJ=100.00
'Path S3818
SFTOF3D
MOVJ C00096 BC00096 VJ=100.00  +MOVJ EC00096 VJ=100.00
MOVL C00097 BC00097 V=666.7  +MOVJ EC00097 VJ=100.00
SMOVL C00098 BC00098 V=166.7  +MOVJ EC00098
SREFP 3 C00099 BC00099  +REFP EC00099
CALL JOB:SEARCH-R1-S13D
SET P062 P006
SFTON3D P062
SMOVL C00100 BC00100 V=166.7  +MOVJ EC00100
SREFP 3 C00101 BC00101  +REFP EC00101
CALL JOB:SEARCH-R1-S13D
SET P062 P006
SFTON3D P062
SMOVL C00102 BC00102 V=166.7  +MOVJ EC00102
SFTOF3D
MOVL C00103 BC00103 V=666.7  +MOVJ EC00103 VJ=100.00
MOVL C00104 BC00104 V=1000.0  +MOVJ EC00104 VJ=100.00
MOVJ C00105 BC00105 VJ=100.00  +MOVJ EC00105 VJ=100.00
MOVJ C00106 BC00106 VJ=100.00  +MOVJ EC00106 VJ=100.00
MOVJ C00107 BC00107 VJ=100.00  +MOVJ EC00107 VJ=100.00
SMOVL C00108 BC00108 V=100.0  +MOVJ EC00108
SREFP 3 C00109 BC00109  +REFP EC00109
CALL JOB:SEARCH-R1-S13D
SET P100 P006
SFTON3D P100
SMOVL C00110 BC00110 V=166.7  +MOVJ EC00110
SREFP 3 C00111 BC00111  +REFP EC00111
CALL JOB:SEARCH-R1-S13D
SET P100 P006
SFTON3D P100
SMOVL C00112 BC00112 V=166.7  +MOVJ EC00112
SMOVL C00113 BC00113 V=250.0  +MOVJ EC00113
SMOVL C00114 BC00114 V=133.3  +MOVJ EC00114
SREFP 3 C00115 BC00115  +REFP EC00115
CALL JOB:SEARCH-R1-S13D
SET P100 P006
SFTON3D P100
SMOVL C00116 BC00116 V=166.7  +MOVJ EC00116
SFTOF3D
MOVJ C00117 BC00117 VJ=100.00  +MOVJ EC00117 VJ=100.00
'
MOVJ C00118 BC00118 VJ=100.00  +MOVJ EC00118 VJ=100.00
MOVJ C00119 BC00119 VJ=100.00  +MOVJ EC00119 VJ=100.00
'Path S3819
SFTOF3D
MOVJ C00120 BC00120 VJ=100.00  +MOVJ EC00120 VJ=100.00
MOVL C00121 BC00121 V=400.0  +MOVJ EC00121 VJ=100.00
SMOVL C00122 BC00122 V=133.3  +MOVJ EC00122
SREFP 3 C00123 BC00123  +REFP EC00123
CALL JOB:SEARCH-R1-S13D
SET P063 P006
SFTON3D P063
SMOVL C00124 BC00124 V=166.7  +MOVJ EC00124
SREFP 3 C00125 BC00125  +REFP EC00125
CALL JOB:SEARCH-R1-S13D
SET P063 P006
SFTON3D P063
SMOVL C00126 BC00126 V=166.7  +MOVJ EC00126
MOVL C00127 BC00127 V=666.7  +MOVJ EC00127 VJ=100.00
MOVL C00128 BC00128 V=1000.0  +MOVJ EC00128 VJ=100.00
'Path S3820
SFTOF3D
MOVJ C00129 BC00129 VJ=100.00  +MOVJ EC00129 VJ=100.00
MOVL C00130 BC00130 V=666.7  +MOVJ EC00130 VJ=100.00
SMOVL C00131 BC00131 V=133.3  +MOVJ EC00131
SREFP 3 C00132 BC00132  +REFP EC00132
CALL JOB:SEARCH-R1-S13D
SET P053 P006
SFTON3D P053
SMOVL C00133 BC00133 V=133.3  +MOVJ EC00133
SREFP 3 C00134 BC00134  +REFP EC00134
CALL JOB:SEARCH-R1-S13D
SET P053 P006
SFTON3D P053
SMOVL C00135 BC00135 V=133.3  +MOVJ EC00135
MOVL C00136 BC00136 V=666.7  +MOVJ EC00136 VJ=100.00
MOVL C00137 BC00137 V=1000.0  +MOVJ EC00137 VJ=100.00
'Path S3821
SFTOF3D
MOVJ C00138 BC00138 VJ=100.00  +MOVJ EC00138 VJ=100.00
MOVL C00139 BC00139 V=400.0  +MOVJ EC00139 VJ=100.00
SMOVL C00140 BC00140 V=133.3  +MOVJ EC00140
SREFP 3 C00141 BC00141  +REFP EC00141
CALL JOB:SEARCH-R1-S13D
SET P043 P006
SFTON3D P043
SMOVL C00142 BC00142 V=166.7  +MOVJ EC00142
SREFP 3 C00143 BC00143  +REFP EC00143
CALL JOB:SEARCH-R1-S13D
SET P043 P006
SFTON3D P043
SMOVL C00144 BC00144 V=166.7  +MOVJ EC00144
MOVL C00145 BC00145 V=666.7  +MOVJ EC00145 VJ=100.00
MOVL C00146 BC00146 V=1000.0  +MOVJ EC00146 VJ=100.00
'Path S3822
SFTOF3D
MOVJ C00147 BC00147 VJ=100.00  +MOVJ EC00147 VJ=100.00
MOVL C00148 BC00148 V=666.7  +MOVJ EC00148 VJ=100.00
SMOVL C00149 BC00149 V=133.3  +MOVJ EC00149
SREFP 3 C00150 BC00150  +REFP EC00150
CALL JOB:SEARCH-R1-S13D
SET P033 P006
SFTON3D P033
SMOVL C00151 BC00151 V=166.7  +MOVJ EC00151
SREFP 3 C00152 BC00152  +REFP EC00152
CALL JOB:SEARCH-R1-S13D
SET P033 P006
SFTON3D P033
SMOVL C00153 BC00153 V=166.7  +MOVJ EC00153
MOVL C00154 BC00154 V=66.7  +MOVJ EC00154 VJ=100.00
MOVL C00155 BC00155 V=1000.0  +MOVJ EC00155 VJ=100.00
'Path S3823
SFTOF3D
MOVJ C00156 BC00156 VJ=100.00  +MOVJ EC00156 VJ=100.00
MOVL C00157 BC00157 V=666.7  +MOVJ EC00157 VJ=100.00
SMOVL C00158 BC00158 V=133.3  +MOVJ EC00158
SREFP 3 C00159 BC00159  +REFP EC00159
CALL JOB:SEARCH-R1-S13D
SET P023 P006
SFTON3D P023
SMOVL C00160 BC00160 V=133.3  +MOVJ EC00160
SREFP 3 C00161 BC00161  +REFP EC00161
CALL JOB:SEARCH-R1-S13D
SET P023 P006
SFTON3D P023
SMOVL C00162 BC00162 V=133.3  +MOVJ EC00162
MOVL C00163 BC00163 V=400.0  +MOVJ EC00163 VJ=100.00
MOVL C00164 BC00164 V=1000.0  +MOVJ EC00164 VJ=100.00
'
'
'
'Path W3824
SFTOF3D
SFTON3D P043
MOVJ C00165 BC00165 VJ=100.00  +MOVJ EC00165 VJ=100.00
SMOVL C00166 BC00166 V=400.0  +MOVJ EC00166
SMOVL C00167 BC00167 V=166.7 PL=0  +MOVJ EC00167
SREFP 1 C00168 BC00168  +REFP EC00168
SREFP 2 C00169 BC00169  +REFP EC00169
MACRO1 MJ#(0) ARGF9
ARCON
SMOVL C00170 BC00170 V=9.2  +MOVJ EC00170
SMOVL C00171 BC00171 V=9.2  +MOVJ EC00171
SMOVL C00172 BC00172 V=9.2  +MOVJ EC00172
ARCOF
SMOVL C00173 BC00173 V=400.0  +MOVJ EC00173
SMOVL C00174 BC00174 V=1000.0  +MOVJ EC00174
SFTOF3D
'Path W3825
SFTOF3D
SFTON3D P023
MOVJ C00175 BC00175 VJ=100.00  +MOVJ EC00175 VJ=100.00
SMOVL C00176 BC00176 V=400.0  +MOVJ EC00176
SMOVL C00177 BC00177 V=166.7 PL=0  +MOVJ EC00177
SREFP 1 C00178 BC00178  +REFP EC00178
SREFP 2 C00179 BC00179  +REFP EC00179
ARCON
SMOVL C00180 BC00180 V=9.2  +MOVJ EC00180
SMOVL C00181 BC00181 V=9.2  +MOVJ EC00181
SMOVL C00182 BC00182 V=9.2  +MOVJ EC00182
ARCOF
SMOVL C00183 BC00183 V=400.0  +MOVJ EC00183
SMOVL C00184 BC00184 V=1000.0  +MOVJ EC00184
SFTOF3D
'Path W3826
SFTOF3D
SFTON3D P063
MOVJ C00185 BC00185 VJ=100.00  +MOVJ EC00185 VJ=100.00
SMOVL C00186 BC00186 V=400.0  +MOVJ EC00186
SMOVL C00187 BC00187 V=166.7 PL=0  +MOVJ EC00187
SREFP 1 C00188 BC00188  +REFP EC00188
SREFP 2 C00189 BC00189  +REFP EC00189
ARCON
SMOVL C00190 BC00190 V=9.2  +MOVJ EC00190
SMOVL C00191 BC00191 V=9.2  +MOVJ EC00191
SMOVL C00192 BC00192 V=9.2  +MOVJ EC00192
ARCOF
SMOVL C00193 BC00193 V=400.0  +MOVJ EC00193
SMOVL C00194 BC00194 V=1000.0  +MOVJ EC00194
SFTOF3D
'Path W3827
SFTOF3D
SFTON3D P033
MOVJ C00195 BC00195 VJ=100.00  +MOVJ EC00195 VJ=100.00
SMOVL C00196 BC00196 V=400.0  +MOVJ EC00196
SMOVL C00197 BC00197 V=166.7 PL=0  +MOVJ EC00197
SREFP 1 C00198 BC00198  +REFP EC00198
SREFP 2 C00199 BC00199  +REFP EC00199
ARCON
SMOVL C00200 BC00200 V=9.2  +MOVJ EC00200
SMOVL C00201 BC00201 V=9.2  +MOVJ EC00201
SMOVL C00202 BC00202 V=9.2  +MOVJ EC00202
ARCOF
SMOVL C00203 BC00203 V=400.0  +MOVJ EC00203
SMOVL C00204 BC00204 V=1000.0  +MOVJ EC00204
SFTOF3D
'Path W3828
SFTOF3D
SFTON3D P053
MOVJ C00205 BC00205 VJ=100.00  +MOVJ EC00205 VJ=100.00
SMOVL C00206 BC00206 V=400.0  +MOVJ EC00206
SMOVL C00207 BC00207 V=166.7 PL=0  +MOVJ EC00207
SREFP 1 C00208 BC00208  +REFP EC00208
SREFP 2 C00209 BC00209  +REFP EC00209
ARCON
SMOVL C00210 BC00210 V=9.2  +MOVJ EC00210
SMOVL C00211 BC00211 V=9.2  +MOVJ EC00211
SMOVL C00212 BC00212 V=9.2  +MOVJ EC00212
ARCOF
SMOVL C00213 BC00213 V=400.0  +MOVJ EC00213
SMOVL C00214 BC00214 V=1000.0  +MOVJ EC00214
SFTOF3D
MOVJ C00215 BC00215 VJ=100.00  +MOVJ EC00215 VJ=100.00
MOVJ C00216 BC00216 VJ=100.00  +MOVJ EC00216 VJ=100.00
MOVJ C00217 BC00217 VJ=100.00  +MOVJ EC00217 VJ=100.00
'
'Path W3829
SFTOF3D
SFTON3D P042
MOVJ C00218 BC00218 VJ=100.00  +MOVJ EC00218 VJ=100.00
SMOVL C00219 BC00219 V=400.0  +MOVJ EC00219
SFTOF3D
SFTON3D P041
SMOVL C00220 BC00220 V=166.7  +MOVJ EC00220
ARCON
SMOVC C00221 BC00221 V=9.2  +MOVJ EC00221
SMOVC C00222 BC00222 V=9.2  +MOVJ EC00222
SMOVC C00223 BC00223 V=9.2  +MOVJ EC00223
SMOVC C00224 BC00224 V=9.2  +MOVJ EC00224
SFTON3D P042
SMOVC C00225 BC00225 V=9.2  +MOVJ EC00225
SMOVL C00226 BC00226 V=9.2  +MOVJ EC00226
ARCOF
SMOVL C00227 BC00227 V=400.0  +MOVJ EC00227
SMOVL C00228 BC00228 V=1000.0  +MOVJ EC00228
SFTOF3D
'Path W3831
SFTOF3D
SFTON3D P041
MOVJ C00229 BC00229 VJ=100.00  +MOVJ EC00229 VJ=100.00
SMOVL C00230 BC00230 V=666.7  +MOVJ EC00230
SMOVL C00231 BC00231 V=166.7 PL=0  +MOVJ EC00231
SREFP 1 C00232 BC00232  +REFP EC00232
SREFP 2 C00233 BC00233  +REFP EC00233
ARCON
SMOVL C00234 BC00234 V=9.2  +MOVJ EC00234
SMOVL C00235 BC00235 V=9.2  +MOVJ EC00235
SMOVL C00236 BC00236 V=9.2  +MOVJ EC00236
ARCOF
SMOVL C00237 BC00237 V=400.0  +MOVJ EC00237
SMOVL C00238 BC00238 V=1000.0  +MOVJ EC00238
SFTOF3D
MOVJ C00239 BC00239 VJ=100.00  +MOVJ EC00239 VJ=100.00
'
'
MOVJ C00240 BC00240 VJ=100.00  +MOVJ EC00240 VJ=100.00
'Path W3832
SFTOF3D
SFTON3D P022
MOVJ C00241 BC00241 VJ=100.00  +MOVJ EC00241 VJ=100.00
SMOVL C00242 BC00242 V=666.7  +MOVJ EC00242
SMOVL C00243 BC00243 V=166.7 PL=0  +MOVJ EC00243
SREFP 1 C00244 BC00244  +REFP EC00244
SREFP 2 C00245 BC00245  +REFP EC00245
ARCON
SMOVL C00246 BC00246 V=9.2  +MOVJ EC00246
SMOVL C00247 BC00247 V=9.2  +MOVJ EC00247
SMOVL C00248 BC00248 V=9.2  +MOVJ EC00248
SMOVL C00249 BC00249 V=9.2  +MOVJ EC00249
ARCOF
SMOVL C00250 BC00250 V=400.0  +MOVJ EC00250
SMOVL C00251 BC00251 V=1000.0  +MOVJ EC00251
SFTOF3D
'Path W3833
SFTOF3D
SFTON3D P021
MOVJ C00252 BC00252 VJ=100.00  +MOVJ EC00252 VJ=100.00
SMOVL C00253 BC00253 V=666.7  +MOVJ EC00253
SMOVL C00254 BC00254 V=166.7 PL=0  +MOVJ EC00254
SREFP 1 C00255 BC00255  +REFP EC00255
SREFP 2 C00256 BC00256  +REFP EC00256
ARCON
SMOVL C00257 BC00257 V=9.2  +MOVJ EC00257
SMOVL C00258 BC00258 V=9.2  +MOVJ EC00258
SMOVL C00259 BC00259 V=9.2  +MOVJ EC00259
SMOVL C00260 BC00260 V=9.2  +MOVJ EC00260
ARCOF
SMOVL C00261 BC00261 V=400.0  +MOVJ EC00261
SMOVL C00262 BC00262 V=1000.0  +MOVJ EC00262
SFTOF3D
'Path W3834
SFTOF3D
SFTON3D P021
MOVJ C00263 BC00263 VJ=100.00  +MOVJ EC00263 VJ=100.00
SMOVL C00264 BC00264 V=666.7  +MOVJ EC00264
SMOVL C00265 BC00265 V=166.7 PL=0  +MOVJ EC00265
SREFP 1 C00266 BC00266  +REFP EC00266
SREFP 2 C00267 BC00267  +REFP EC00267
ARCON
SMOVL C00268 BC00268 V=9.2  +MOVJ EC00268
SMOVL C00269 BC00269 V=9.2  +MOVJ EC00269
SMOVL C00270 BC00270 V=9.2  +MOVJ EC00270
ARCOF
SMOVL C00271 BC00271 V=400.0  +MOVJ EC00271
SMOVL C00272 BC00272 V=1000.0  +MOVJ EC00272
SFTOF3D
MOVJ C00273 BC00273 VJ=100.00  +MOVJ EC00273 VJ=100.00
'
'
MOVJ C00274 BC00274 VJ=100.00  +MOVJ EC00274 VJ=100.00
'Path W3835
SFTOF3D
SFTON3D P062
MOVJ C00275 BC00275 VJ=100.00  +MOVJ EC00275 VJ=100.00
SMOVL C00276 BC00276 V=666.7  +MOVJ EC00276
SMOVL C00277 BC00277 V=166.7 PL=0  +MOVJ EC00277
SREFP 1 C00278 BC00278  +REFP EC00278
SREFP 2 C00279 BC00279  +REFP EC00279
ARCON
SMOVL C00280 BC00280 V=9.2  +MOVJ EC00280
SMOVL C00281 BC00281 V=9.2  +MOVJ EC00281
SMOVL C00282 BC00282 V=9.2  +MOVJ EC00282
ARCOF
SMOVL C00283 BC00283 V=400.0  +MOVJ EC00283
SMOVL C00284 BC00284 V=1000.0  +MOVJ EC00284
SFTOF3D
'Path W3836
SFTOF3D
SFTON3D P061
MOVJ C00285 BC00285 VJ=100.00  +MOVJ EC00285 VJ=100.00
SMOVL C00286 BC00286 V=666.7  +MOVJ EC00286
SMOVL C00287 BC00287 V=166.7 PL=0  +MOVJ EC00287
SREFP 1 C00288 BC00288  +REFP EC00288
SREFP 2 C00289 BC00289  +REFP EC00289
ARCON
SMOVL C00290 BC00290 V=9.2  +MOVJ EC00290
SMOVL C00291 BC00291 V=9.2  +MOVJ EC00291
SMOVL C00292 BC00292 V=9.2  +MOVJ EC00292
SMOVL C00293 BC00293 V=9.2  +MOVJ EC00293
ARCOF
SMOVL C00294 BC00294 V=400.0  +MOVJ EC00294
SMOVL C00295 BC00295 V=1000.0  +MOVJ EC00295
SFTOF3D
'Path W3837
SFTOF3D
SFTON3D P061
MOVJ C00296 BC00296 VJ=100.00  +MOVJ EC00296 VJ=100.00
SMOVL C00297 BC00297 V=666.7  +MOVJ EC00297
SMOVL C00298 BC00298 V=166.7 PL=0  +MOVJ EC00298
SREFP 1 C00299 BC00299  +REFP EC00299
SREFP 2 C00300 BC00300  +REFP EC00300
ARCON
SMOVL C00301 BC00301 V=9.2  +MOVJ EC00301
SMOVL C00302 BC00302 V=9.2  +MOVJ EC00302
SMOVL C00303 BC00303 V=9.2  +MOVJ EC00303
ARCOF
SMOVL C00304 BC00304 V=400.0  +MOVJ EC00304
SMOVL C00305 BC00305 V=1000.0  +MOVJ EC00305
SFTOF3D
MOVJ C00306 BC00306 VJ=100.00  +MOVJ EC00306 VJ=100.00
'
'
MOVJ C00307 BC00307 VJ=100.00  +MOVJ EC00307 VJ=100.00
'Path W3838
SFTOF3D
SFTON3D P032
MOVJ C00308 BC00308 VJ=100.00  +MOVJ EC00308 VJ=100.00
SMOVL C00309 BC00309 V=666.7  +MOVJ EC00309
SMOVL C00310 BC00310 V=166.7 PL=0  +MOVJ EC00310
SREFP 1 C00311 BC00311  +REFP EC00311
SREFP 2 C00312 BC00312  +REFP EC00312
ARCON
SMOVL C00313 BC00313 V=9.2  +MOVJ EC00313
SMOVL C00314 BC00314 V=9.2  +MOVJ EC00314
SMOVL C00315 BC00315 V=9.2  +MOVJ EC00315
SMOVL C00316 BC00316 V=9.2  +MOVJ EC00316
ARCOF
SMOVL C00317 BC00317 V=400.0  +MOVJ EC00317
SMOVL C00318 BC00318 V=1000.0  +MOVJ EC00318
SFTOF3D
'Path W3839
SFTOF3D
SFTON3D P031
MOVJ C00319 BC00319 VJ=100.00  +MOVJ EC00319 VJ=100.00
SMOVL C00320 BC00320 V=666.7  +MOVJ EC00320
SMOVL C00321 BC00321 V=166.7 PL=0  +MOVJ EC00321
SREFP 1 C00322 BC00322  +REFP EC00322
SREFP 2 C00323 BC00323  +REFP EC00323
ARCON
SMOVL C00324 BC00324 V=9.2  +MOVJ EC00324
SMOVL C00325 BC00325 V=9.2  +MOVJ EC00325
SMOVL C00326 BC00326 V=9.2  +MOVJ EC00326
SMOVL C00327 BC00327 V=9.2  +MOVJ EC00327
ARCOF
SMOVL C00328 BC00328 V=400.0  +MOVJ EC00328
SMOVL C00329 BC00329 V=1000.0  +MOVJ EC00329
SFTOF3D
'Path W3840
SFTOF3D
SFTON3D P031
MOVJ C00330 BC00330 VJ=100.00  +MOVJ EC00330 VJ=100.00
SMOVL C00331 BC00331 V=666.7  +MOVJ EC00331
SMOVL C00332 BC00332 V=166.7 PL=0  +MOVJ EC00332
SREFP 1 C00333 BC00333  +REFP EC00333
SREFP 2 C00334 BC00334  +REFP EC00334
ARCON
SMOVL C00335 BC00335 V=9.2  +MOVJ EC00335
SMOVL C00336 BC00336 V=9.2  +MOVJ EC00336
SMOVL C00337 BC00337 V=9.2  +MOVJ EC00337
ARCOF
SMOVL C00338 BC00338 V=400.0  +MOVJ EC00338
SMOVL C00339 BC00339 V=1000.0  +MOVJ EC00339
SFTOF3D
MOVJ C00340 BC00340 VJ=100.00  +MOVJ EC00340 VJ=100.00
'
'
MOVJ C00341 BC00341 VJ=100.00  +MOVJ EC00341 VJ=100.00
'Path W3841
SFTOF3D
SFTON3D P052
MOVJ C00342 BC00342 VJ=100.00  +MOVJ EC00342 VJ=100.00
SMOVL C00343 BC00343 V=666.7  +MOVJ EC00343
SMOVL C00344 BC00344 V=166.7 PL=0  +MOVJ EC00344
SREFP 1 C00345 BC00345  +REFP EC00345
SREFP 2 C00346 BC00346  +REFP EC00346
ARCON
SMOVL C00347 BC00347 V=9.2  +MOVJ EC00347
SMOVL C00348 BC00348 V=9.2  +MOVJ EC00348
SMOVL C00349 BC00349 V=9.2  +MOVJ EC00349
SMOVL C00350 BC00350 V=9.2  +MOVJ EC00350
ARCOF
SMOVL C00351 BC00351 V=400.0  +MOVJ EC00351
SMOVL C00352 BC00352 V=1000.0  +MOVJ EC00352
SFTOF3D
'Path W3842
SFTOF3D
SFTON3D P051
MOVJ C00353 BC00353 VJ=100.00  +MOVJ EC00353 VJ=100.00
SMOVL C00354 BC00354 V=666.7  +MOVJ EC00354
SMOVL C00355 BC00355 V=166.7 PL=0  +MOVJ EC00355
SREFP 1 C00356 BC00356  +REFP EC00356
SREFP 2 C00357 BC00357  +REFP EC00357
ARCON
SMOVL C00358 BC00358 V=9.2  +MOVJ EC00358
SMOVL C00359 BC00359 V=9.2  +MOVJ EC00359
SMOVL C00360 BC00360 V=9.2  +MOVJ EC00360
SMOVL C00361 BC00361 V=9.2  +MOVJ EC00361
SMOVL C00362 BC00362 V=9.2  +MOVJ EC00362
ARCOF
SMOVL C00363 BC00363 V=400.0  +MOVJ EC00363
SMOVL C00364 BC00364 V=1000.0  +MOVJ EC00364
SFTOF3D
'Path W3843
SFTOF3D
SFTON3D P051
MOVJ C00365 BC00365 VJ=100.00  +MOVJ EC00365 VJ=100.00
SMOVL C00366 BC00366 V=666.7  +MOVJ EC00366
SMOVL C00367 BC00367 V=166.7 PL=0  +MOVJ EC00367
SREFP 1 C00368 BC00368  +REFP EC00368
SREFP 2 C00369 BC00369  +REFP EC00369
ARCON
SMOVL C00370 BC00370 V=9.2  +MOVJ EC00370
SMOVL C00371 BC00371 V=9.2  +MOVJ EC00371
SMOVL C00372 BC00372 V=9.2  +MOVJ EC00372
ARCOF
SMOVL C00373 BC00373 V=400.0  +MOVJ EC00373
SMOVL C00374 BC00374 V=1000.0  +MOVJ EC00374
SFTOF3D
MOVJ C00375 BC00375 VJ=100.00  +MOVJ EC00375 VJ=100.00
MOVJ C00376 BC00376 VJ=100.00  +MOVJ EC00376 VJ=100.00
SFTON3D P100
SMOVL C00377 BC00377 V=166.7 PL=0  +MOVJ EC00377
SREFP 1 C00378 BC00378  +REFP EC00378
SREFP 2 C00379 BC00379  +REFP EC00379
ARCON
SWVON WEV#(102)
SMOVL C00380 BC00380 V=7.5  +MOVJ EC00380
SMOVL C00381 BC00381 V=7.5  +MOVJ EC00381
ARCOF
SWVOF
SMOVL C00382 BC00382 V=250.0  +MOVJ EC00382
SMOVL C00383 BC00383 V=250.0  +MOVJ EC00383
SMOVL C00384 BC00384 V=333.3  +MOVJ EC00384
SFTON3D P100
MACRO1 MJ#(0) ARGF14
SMOVL C00385 BC00385 V=133.3  +MOVJ EC00385
ARCON
SWVON WEV#(66)
SMOVL C00386 BC00386 V=10.8  +MOVJ EC00386
SMOVL C00387 BC00387 V=10.8  +MOVJ EC00387
SMOVL C00388 BC00388 V=10.8  +MOVJ EC00388
ARCOF
SWVOF
SFTOF3D
SMOVL C00389 BC00389 V=333.3  +MOVJ EC00389
MOVJ C00390 BC00390 VJ=100.00  +MOVJ EC00390 VJ=100.00
'
END
